# EPICS autosave request: softGlueApp/Db/softGlue_SignalShow_settings.req
$(P)$(H)ReadRateON.SCAN
$(P)$(H)ReadRateOFF.SCAN
